PROGRAM A_Program
VAR
	i : UINT;
	x : LREAL;
	x_inc : LREAL := 0.0001;
END_VAR

FOR i := 0 TO 1000 DO
	x := x + x_inc;
END_FOR

END_PROGRAM

(* stored: Version 1.1.0.1, ProductVersion 3.1.4025.12
   POU A_Program: Id {bf40f532-2487-47cf-b1c4-3c529584f388}, SpecialFunc None *)
